PROGRAM MAIN
VAR
END_VAR

END_PROGRAM

(* stored: Version 1.1.0.1, ProductVersion 3.1.4024.12
   POU MAIN: Id {f7299d14-1675-426f-a592-4bcc09daeca7}, SpecialFunc None *)
